ABB RobotStudio station: saddlewelding_table.rspag

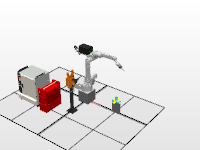
--- station ---
Station Final_1520_table (saved by RobotStudio 7.0.8743.626)
Controller 1520_simple_table_base, task T_ROB1: task frame (RAPID world) sits at (0, 0, 350) mm in the station
Controller 1520_simple_table_base
  mechanical unit ROB_1: IRB1520ID_4_150__02, 6 joints, base frame (0, 0, 0) mm
Layout (positions relative to the parent item):
  - IRB1520ID_4_150__02 [mechanism, from Robots\IRB1520ID_4_150_G_02.rslib] at (0, 0, 350) mm; joint values [0, 0, 0, 0, 0.5236, 0] (rad or m)
  - Binzel_ID_22 [mechanism, from Tools\Binzel_ID_22.rslib] at (1056.21, 0, 1493) mm, rotated rx 180 ry 60 rz 180 deg
  - base [part]
  - saddle_simple_tpipe [part] at (1025, 0, 375) mm, rotated rx 90 ry 0 rz 0 deg
  - table [part] at (1025, 0, 0) mm, rotated rx 0 ry 0 rz 90 deg
  - IRC5_Singel-Cabinet [part, from Equipment\IRC5_Singel-Cabinet.rslib] at (-1225.42, -1000, 100) mm, rotated rx 90 ry 0 rz 0 deg
  - Fronius_VR1500 [part, from Equipment\Fronius_VR1500.rslib] at (-205.78, 25.28, 165.99) mm
  - Fronius_TPS4000_rev0 [part, from Equipment\Fronius_TPS4000.rslib] at (-617.24, -872.21, 0) mm, rotated rx 0 ry 0 rz 180 deg
  - torch_cleaner_binzel [graphiccomponentgroup, from Equipment\Torch Cleaner Binzel.rslib] at (0, -659.93, 0) mm
    - Body 1 [part, from Equipment\Torch Cleaner Binzel.rslib]
    - Body 2 [part, from Equipment\Torch Cleaner Binzel.rslib]
    - Body 3 [part, from Equipment\Torch Cleaner Binzel.rslib]
    - Body 4 [part, from Equipment\Torch Cleaner Binzel.rslib]
    - Body 5 [part, from Equipment\Torch Cleaner Binzel.rslib]
    - Body 6 [part, from Equipment\Torch Cleaner Binzel.rslib]
    - Body 7 [part, from Equipment\Torch Cleaner Binzel.rslib]
    - Body 8 [part, from Equipment\Torch Cleaner Binzel.rslib]
    - Body 9 [part, from Equipment\Torch Cleaner Binzel.rslib]
    - Body 10 [part, from Equipment\Torch Cleaner Binzel.rslib]
    - Body 11 [part, from Equipment\Torch Cleaner Binzel.rslib]
    - Body 12 [part, from Equipment\Torch Cleaner Binzel.rslib]
Attachment: Binzel_ID_22 is attached to IRB1520ID_4_150__02 / Link6
Attachment: Fronius_VR1500 is attached to IRB1520ID_4_150__02 / Link3

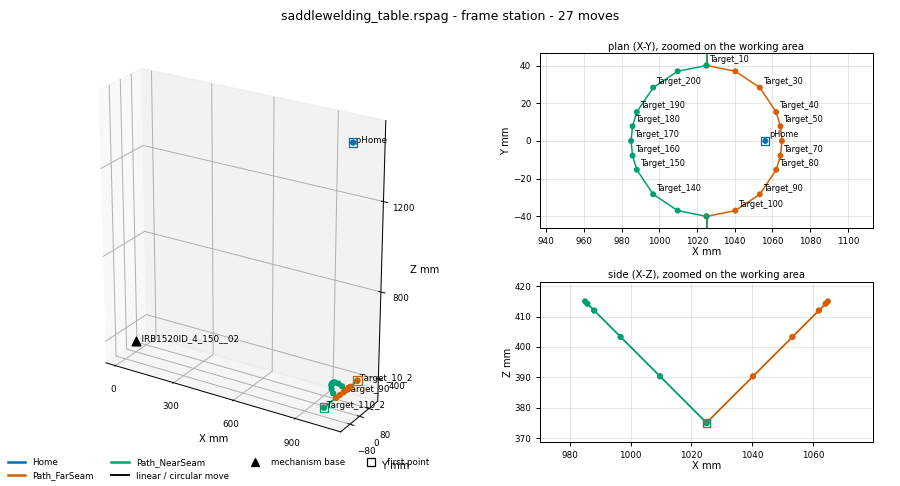
[picture p0: tool path of saddlewelding_table.rspag in frame station, 27 of 27 moves have a stored position in this frame; points joined in program order, loops and branches not executed]
--- Backups/1520_simple_table_base/RAPID/TASK1/PROGMOD/CalibData.mod ---
MODULE CalibData
	PERS tooldata tWeldGun:=[TRUE,[[49.841566361,0,372.194826196],[0.981627183,0,0.190808995,0]],[2,[0,0,100],[0,1,0,0],0,0,0]];
	TASK PERS wobjdata Workobject_1:=[FALSE,TRUE,"",[[1275,0,-15],[1,0,0,0]],[[0,0,0],[1,0,0,0]]];
ENDMODULE

--- Backups/1520_simple_table_base/RAPID/TASK1/PROGMOD/Module1.mod ---
MODULE Module1
	CONST robtarget Target_20:=[[-234.692662705,36.9551813,55.307337295],[0.301754825,0.232815701,-0.741273461,0.552498444],[0,0,0,0],[9E+09,9E+09,9E+09,9E+09,9E+09,9E+09]];
	CONST robtarget Target_30:=[[-221.715728753,28.284271247,68.284271247],[0.339851143,0.175919897,-0.820473238,0.424708201],[0,0,0,0],[9E+09,9E+09,9E+09,9E+09,9E+09,9E+09]];
	CONST robtarget Target_40:=[[-213.0448187,15.307337295,76.9551813],[0.401835396,0.091255347,-0.877471606,0.245447259],[0,0,0,0],[9E+09,9E+09,9E+09,9E+09,9E+09,9E+09]];
	CONST robtarget Target_50:=[[-210.768588784,7.803612881,79.231411216],[0.387785125,0.051100945,-0.911559828,0.126767777],[0,0,0,0],[9E+09,9E+09,9E+09,9E+09,9E+09,9E+09]];
	CONST robtarget Target_60:=[[-210,0,80],[0.382683432,0,-0.923879533,0],[0,0,0,0],[9E+09,9E+09,9E+09,9E+09,9E+09,9E+09]];
	CONST robtarget Target_70:=[[-210.768588784,-7.803612881,79.231411216],[0.387785125,-0.051100945,-0.911559828,-0.126767777],[0,0,0,0],[9E+09,9E+09,9E+09,9E+09,9E+09,9E+09]];
	CONST robtarget Target_80:=[[-213.0448187,-15.307337295,76.9551813],[0.401835396,-0.091255347,-0.877471606,-0.245447259],[0,0,0,0],[9E+09,9E+09,9E+09,9E+09,9E+09,9E+09]];
	CONST robtarget Target_90:=[[-221.715728753,-28.284271247,68.284271247],[0.339851143,-0.175919897,-0.820473238,-0.424708201],[0,0,0,0],[9E+09,9E+09,9E+09,9E+09,9E+09,9E+09]];
	CONST robtarget Target_100:=[[-234.692662705,-36.9551813,55.307337295],[0.301754825,-0.232815702,-0.741273461,-0.552498444],[0,0,0,0],[9E+09,9E+09,9E+09,9E+09,9E+09,9E+09]];
	CONST robtarget Target_110:=[[-250,-40,40],[0.27059805,-0.27059805,-0.653281483,-0.653281482],[0,0,0,0],[9E+09,9E+09,9E+09,9E+09,9E+09,9E+09]];
	CONST robtarget Target_120:=[[-250,-40,40],[0.653281482,-0.653281483,-0.27059805,-0.27059805],[0,0,0,0],[9E+09,9E+09,9E+09,9E+09,9E+09,9E+09]];
	CONST robtarget Target_130:=[[-265.307337295,-36.9551813,55.307337295],[0.552498444,-0.741273461,-0.232815702,-0.301754825],[0,0,0,0],[9E+09,9E+09,9E+09,9E+09,9E+09,9E+09]];
	CONST robtarget Target_140:=[[-278.284271247,-28.284271247,68.284271247],[0.424708201,-0.820473238,-0.175919897,-0.339851143],[0,0,0,0],[9E+09,9E+09,9E+09,9E+09,9E+09,9E+09]];
	CONST robtarget Target_150:=[[-286.9551813,-15.307337295,76.9551813],[0.245447259,-0.877471606,-0.091255347,-0.401835396],[0,0,0,0],[9E+09,9E+09,9E+09,9E+09,9E+09,9E+09]];
	CONST robtarget Target_160:=[[-289.231411216,-7.803612881,79.231411216],[0.126767777,-0.911559828,-0.051100945,-0.387785125],[0,0,0,0],[9E+09,9E+09,9E+09,9E+09,9E+09,9E+09]];
	CONST robtarget Target_170:=[[-290,0,80],[0,0.923879533,0,0.382683432],[0,0,0,0],[9E+09,9E+09,9E+09,9E+09,9E+09,9E+09]];
	CONST robtarget Target_180:=[[-289.231411216,7.803612881,79.231411216],[0.126767777,0.911559828,-0.051100945,0.387785125],[0,0,0,0],[9E+09,9E+09,9E+09,9E+09,9E+09,9E+09]];
	CONST robtarget Target_190:=[[-286.9551813,15.307337295,76.9551813],[0.245447259,0.877471606,-0.091255347,0.401835396],[0,0,0,0],[9E+09,9E+09,9E+09,9E+09,9E+09,9E+09]];
	CONST robtarget Target_200:=[[-278.284271247,28.284271247,68.284271247],[0.424708201,0.820473238,-0.175919897,0.339851143],[0,0,0,0],[9E+09,9E+09,9E+09,9E+09,9E+09,9E+09]];
	CONST robtarget Target_210:=[[-265.307337295,36.9551813,55.307337295],[0.552498444,0.741273461,-0.232815702,0.301754825],[0,0,0,0],[9E+09,9E+09,9E+09,9E+09,9E+09,9E+09]];
	CONST robtarget Target_220:=[[-250,40,40],[0.653281482,0.653281483,-0.27059805,0.27059805],[0,0,0,0],[9E+09,9E+09,9E+09,9E+09,9E+09,9E+09]];
	CONST robtarget Target_230:=[[-282.453870239,-23.382606923,72.453870239],[0.36908745,-0.817925816,-0.11640561,-0.425701242],[0,0,0,0],[9E+09,9E+09,9E+09,9E+09,9E+09,9E+09]];
	CONST robtarget Target_240:=[[-286.842532921,-15.576513344,76.842532921],[0.249627409,-0.875865985,-0.092436435,-0.40249278],[0,0,0,0],[9E+09,9E+09,9E+09,9E+09,9E+09,9E+09]];
	CONST robtarget Target_250:=[[-289.492720807,-6.350197107,79.492720807],[0.103339371,-0.915697289,-0.042043632,-0.38607225],[0,0,0,0],[9E+09,9E+09,9E+09,9E+09,9E+09,9E+09]];
	CONST robtarget Target_260:=[[-289.838896322,3.586410435,79.838896322],[0.05850504,0.9212589,-0.024095941,0.383768922],[0,0,0,0],[9E+09,9E+09,9E+09,9E+09,9E+09,9E+09]];
	CONST robtarget Target_270:=[[-287.790501577,13.110224658,77.790501577],[0.211127225,0.889602963,-0.080867869,0.396852934],[0,0,0,0],[9E+09,9E+09,9E+09,9E+09,9E+09,9E+09]];
	CONST robtarget Target_280:=[[-283.824537222,21.351830875,73.824537222],[0.338236757,0.835161577,-0.112262157,0.418925106],[0,0,0,0],[9E+09,9E+09,9E+09,9E+09,9E+09,9E+09]];
	CONST robtarget Target_290:=[[-278.562833915,28.002937681,68.562833915],[0.439678809,0.772214203,-0.11915461,0.442910768],[0,0,0,0],[9E+09,9E+09,9E+09,9E+09,9E+09,9E+09]];
	CONST robtarget Target_300:=[[-272.483009037,33.083444571,62.483009037],[0.521308907,0.707587067,-0.108046549,0.464632661],[0,0,0,0],[9E+09,9E+09,9E+09,9E+09,9E+09,9E+09]];
	CONST robtarget Target_310:=[[-265.898978741,36.704529353,55.898978741],[0.58859417,0.643472913,-0.084415573,0.482051372],[0,0,0,0],[9E+09,9E+09,9E+09,9E+09,9E+09,9E+09]];
	CONST robtarget Target_320:=[[-259.017319759,38.970346988,49.017319759],[0.645433608,0.580218539,-0.051773745,0.494045933],[0,0,0,0],[9E+09,9E+09,9E+09,9E+09,9E+09,9E+09]];
	CONST robtarget Target_330:=[[-251.98508554,39.950712577,41.98508554],[0.694474459,0.51755125,-0.012188894,0.499697268],[0,0,0,0],[9E+09,9E+09,9E+09,9E+09,9E+09,9E+09]];
	CONST robtarget Target_10:=[[-250,40,40],[0.27059805,0.27059805,-0.653281483,0.653281482],[0,0,0,0],[9E+09,9E+09,9E+09,9E+09,9E+09,9E+09]];
	CONST robtarget pHome:=[[1056.205080757,0,1143],[0.5,0,0.866025404,0],[0,0,0,0],[9E+09,9E+09,9E+09,9E+09,9E+09,9E+09]];
	CONST robtarget Target_10_2:=[[-250,140,40],[0.27059805,0.27059805,-0.653281483,0.653281482],[0,0,0,0],[9E+09,9E+09,9E+09,9E+09,9E+09,9E+09]];
	CONST robtarget Target_110_2:=[[-250,-140,40],[0.27059805,-0.27059805,-0.653281483,-0.653281482],[0,0,0,0],[9E+09,9E+09,9E+09,9E+09,9E+09,9E+09]];
	CONST robtarget Target_120_2:=[[-250,-140,40],[0.653281482,-0.653281483,-0.27059805,-0.27059805],[0,0,0,0],[9E+09,9E+09,9E+09,9E+09,9E+09,9E+09]];
	CONST robtarget Target_220_2:=[[-250,140,40],[0.653281482,0.653281483,-0.27059805,0.27059805],[0,0,0,0],[9E+09,9E+09,9E+09,9E+09,9E+09,9E+09]];
    !***********************************************************
    !
    ! Module:  Module1
    !
    ! Description:
    !   <Insert description here>
    !
    ! Author: firmi
    !
    ! Version: 1.0
    !
    !***********************************************************


    !***********************************************************
    !
    ! Procedure main
    !
    !   This is the entry point of your program
    !


    !***********************************************************
    PROC main()
        !Add your code here
        Home;
        Path_FarSeam;
        !Home;
        Path_NearSeam;
        Home;
    ENDPROC

	PROC Home()
	    MoveJ pHome,v400,z0,tWeldGun\WObj:=wobj0;
	ENDPROC
	PROC Path_FarSeam()
	    MoveL Target_10_2,v400,z0,tWeldGun\WObj:=Workobject_1;
	    MoveL Target_10,v50,z0,tWeldGun\WObj:=Workobject_1;
	    MoveL Target_20,v50,z0,tWeldGun\WObj:=Workobject_1;
	    MoveL Target_30,v50,z0,tWeldGun\WObj:=Workobject_1;
	    MoveL Target_40,v50,z0,tWeldGun\WObj:=Workobject_1;
	    MoveL Target_50,v50,z0,tWeldGun\WObj:=Workobject_1;
	    MoveL Target_60,v50,z0,tWeldGun\WObj:=Workobject_1;
	    MoveL Target_70,v50,z0,tWeldGun\WObj:=Workobject_1;
	    MoveL Target_80,v50,z0,tWeldGun\WObj:=Workobject_1;
	    MoveL Target_90,v50,z0,tWeldGun\WObj:=Workobject_1;
	    MoveL Target_100,v50,z0,tWeldGun\WObj:=Workobject_1;
	    MoveL Target_110,v50,z0,tWeldGun\WObj:=Workobject_1;
	    MoveL Target_110_2,v50,z0,tWeldGun\WObj:=Workobject_1;
	ENDPROC
	PROC Path_NearSeam()
	    MoveL Target_120_2,v50,z0,tWeldGun\WObj:=Workobject_1;
	    MoveL Target_120,v50,z0,tWeldGun\WObj:=Workobject_1;
	    MoveL Target_130,v50,z0,tWeldGun\WObj:=Workobject_1;
	    MoveL Target_140,v50,z0,tWeldGun\WObj:=Workobject_1;
	    MoveL Target_150,v50,z0,tWeldGun\WObj:=Workobject_1;
	    MoveL Target_160,v50,z0,tWeldGun\WObj:=Workobject_1;
	    MoveL Target_170,v50,z0,tWeldGun\WObj:=Workobject_1;
	    MoveL Target_180,v50,z0,tWeldGun\WObj:=Workobject_1;
	    MoveL Target_190,v50,z0,tWeldGun\WObj:=Workobject_1;
	    MoveL Target_200,v50,z0,tWeldGun\WObj:=Workobject_1;
	    MoveL Target_210,v50,z0,tWeldGun\WObj:=Workobject_1;
	    MoveL Target_220,v50,z0,tWeldGun\WObj:=Workobject_1;
	    MoveL Target_220_2,v50,z0,tWeldGun\WObj:=Workobject_1;
	ENDPROC
ENDMODULE
